Universal Robots PolyScope program: Test ur5c.urp

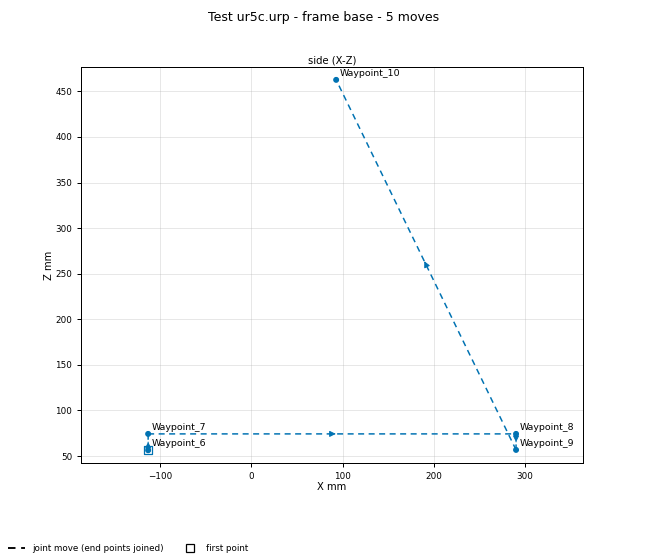
[picture p0: tool path of Test ur5c.urp in frame base, 5 of 5 moves have a stored position in this frame; points joined in program order, loops and branches not executed]
Program Test ur5c (installation=default directory=/programs/usbdisk/NoodleBotSoftware createdIn=3.12.1.90940 lastSavedIn=3.12.1.90940 robotSerialNumber=2017354841)
Calibrated DH parameters: a=[0.000094, -0.006117, -0.382762, 0.000086, 0.000044, 0]; d=[0.089236, 217.751846, -204.357806, -13.283746, 0.094902, 0.082641]; alpha=[1.57017, 0.001953, -0.006493, 1.570192, -1.570543, 0]; deltaTheta=[0.000036, 1.556386, -1.779789, 0.223359, -0.000014, -0.000001]
Robot Program (runOnlyOnce=false)
  MoveL speed 1000 mm/s, acceleration 1200 mm/s^2 (useActiveTCP=true) feature=Base
    Waypoint Waypoint_6: TCP in base x=-113.258 y=-352.946 z=56.387 mm, rx=2.4743 ry=-1.0833 rz=-0.457 rad; joints [69.144, -107, 145.455, 208.353, 250.31, 22.147] deg; flange x=-30.393 y=-310.636 z=218.136 mm, rx=-1.105 ry=-2.5237 rz=0.5696 rad
    MoveJ speed 60 deg/s, acceleration 80 deg/s^2 (useActiveTCP=true)
      Waypoint Waypoint_7: TCP in base x=-113.258 y=-352.951 z=74.319 mm, rx=2.4743 ry=-1.0834 rz=-0.4569 rad; joints [69.139, -109.46, 143.632, 212.639, 250.292, 22.157] deg; flange x=-30.393 y=-310.636 z=236.077 mm, rx=-1.105 ry=-2.5237 rz=0.5696 rad
    MoveJ speed 60 deg/s, acceleration 80 deg/s^2 (useActiveTCP=true)
      Waypoint Waypoint_8: TCP in base x=290.243 y=-352.982 z=74.321 mm, rx=2.4743 ry=-1.0834 rz=-0.4569 rad; joints [131.849, -82.771, 111.76, 249.375, 240.883, 91.284] deg; flange x=373.08 y=-310.636 z=236.077 mm, rx=-1.105 ry=-2.5237 rz=0.5696 rad
    MoveJ speed 60 deg/s, acceleration 80 deg/s^2 (useActiveTCP=true)
      Waypoint Waypoint_9: TCP in base x=290.239 y=-353.007 z=56.761 mm, rx=2.4742 ry=-1.0833 rz=-0.4568 rad; joints [131.853, -81.474, 113.224, 246.609, 240.886, 91.271] deg; flange x=373.08 y=-310.636 z=218.448 mm, rx=-1.105 ry=-2.5237 rz=0.5696 rad
    URCap RG2 (RG - On Robot, OnRobot A/S) dataModel(depthCompensate=false, force=40, payload=0.0, width=85, name=RG2(85))
    MoveJ speed 60 deg/s, acceleration 80 deg/s^2 (useActiveTCP=true)
      Waypoint Waypoint_10: TCP in base x=92.943 y=-353.109 z=462.615 mm, rx=1.1692 ry=-1.2408 rz=1.1709 rad; joints [88.542, -137.017, 138.651, 178.588, 268.345, 89.997] deg; flange x=103.1 y=-166.785 z=463.289 mm, rx=1.2543 ry=1.1819 rz=-1.2438 rad
